Yaskawa INFORM job: R2_W53-A5(180,0)AWOK.JBI

/JOB
//NAME R2_W53-A5(180,0)AWOK
///FOLDERNAME AWOK
//POS
///NPOS 32,32,0,2,0,0
///TOOL 0
///POSTYPE PULSE
///PULSE
C00000=78189,-67986,-96830,-10467,37806,-7797
C00001=92440,-137165,-107216,-20191,-1154,-30432
C00002=105503,-62969,-89657,-20228,86421,-49842
C00003=110518,-93811,-72284,-25294,103379,-67006
C00004=109543,-97011,-70118,-25208,100377,-66720
C00005=109125,-98154,-69170,-25203,99187,-66619
C00006=109125,-97062,-67033,-25140,98501,-66471
C00007=109125,-98154,-69170,-25203,99187,-66619
C00008=109271,-97171,-69065,-25206,99632,-66661
C00009=108845,-100765,-70348,-25219,98541,-66586
C00010=109271,-97171,-69065,-25206,99632,-66661
C00011=102810,-100484,-71733,-21889,96863,-67504
C00012=105287,-101169,-71975,-21344,97318,-66684
C00013=102810,-100484,-71733,-21889,96863,-67504
C00014=103151,-99431,-72768,-21891,98051,-67597
C00015=103951,-96443,-75155,-21958,101060,-67861
C00016=107257,-100648,-73272,-10850,107469,-69930
C00017=107258,-98768,-69563,-10763,106175,-69811
C00018=112732,-102414,-73458,-8827,107350,-67938
C00019=107259,-98817,-69673,-10765,106216,-69815
C00020=107581,-95618,-67198,-10659,106378,-69713
C00021=107132,-98744,-68135,-10755,105306,-69778
C00022=106572,-95477,-62214,-34043,93376,-79177
C00023=105781,-95731,-62292,-31308,97836,-75763
C00024=108056,-94926,-62112,-24163,105722,-68769
C00025=107208,-94572,-61089,-27775,101795,-84365
C00026=107266,-95021,-62493,-27833,102377,-84485
C00027=107266,-96693,-65652,-27971,103342,-84724
C00028=122843,-112109,-94588,-24450,117159,-81729
C00029=129835,-134677,-103725,-23924,94621,-78436
C00030=118025,-147103,-122296,-20754,32567,-81607
C00031=61610,-147103,-122296,-20754,32567,-81607
BC00000=191480,239490,1075165
BC00001=211047,195744,1075167
BC00002=219137,147036,1075169
BC00003=237082,38982,1075175
BC00004=237082,38982,1075175
BC00005=237082,38982,1075175
BC00006=237082,38982,1075175
BC00007=237082,38982,1075175
BC00008=237082,38982,1075175
BC00009=237082,38982,1075175
BC00010=237082,38982,1075175
BC00011=237082,38982,1075175
BC00012=237082,38982,1075175
BC00013=237082,38982,1075175
BC00014=237082,38982,1075175
BC00015=237082,38982,1075175
BC00016=264111,22038,1075175
BC00017=262937,27424,1075175
BC00018=262467,29578,1075175
BC00019=262467,29578,1075175
BC00020=262467,29578,1075175
BC00021=262467,29578,1075175
BC00022=226039,41359,1075175
BC00023=234841,33538,1075175
BC00024=257071,26439,1075171
BC00025=249909,32280,1075175
BC00026=249045,29914,1075175
BC00027=246884,23997,1075175
BC00028=246884,23997,1075175
BC00029=246884,23997,1075175
BC00030=246884,78765,1075175
BC00031=208302,298254,1075175
///POSTYPE BASE
///RECTAN
///RCONF 0,0,0,0,0,0,0,0,0,0,0,0,0,0,0,0,0,0,0,0,0,0,0,0
P00006=0.222,-3.123,-1.508,0.0000,0.0000,0.0000
P00023=0.143,-0.036,0.682,0.0000,0.0000,0.0000
//INST
///DATE 2023/11/16 10:54
///ATTR SC,RW
///GROUP1 RB1,BS1
NOP
'r2_W53-A5(180,0)
'Path S1074
MOVJ C00000 BC00000 VJ=20.00
SFTOF
MOVJ C00001 BC00001 VJ=20.00
MOVJ C00002 BC00002 VJ=20.00
MOVJ C00003 BC00003 VJ=20.00
MOVL C00004 BC00004 V=100.0
MOVL C00005 BC00005 V=60.0
REFP 3 C00006 BC00006
CALL JOB:SEARCH-R1
SET P023 P006
SFTON P023
MOVL C00007 BC00007 V=60.0
MOVL C00008 BC00008 V=60.0
REFP 3 C00009 BC00009
CALL JOB:SEARCH-R1
SET P023 P006
SFTON P023
MOVL C00010 BC00010 V=60.0
MOVL C00011 BC00011 V=60.0
REFP 3 C00012 BC00012
CALL JOB:SEARCH-R1
SET P023 P006
SFTON P023
MOVL C00013 BC00013 V=60.0
MOVL C00014 BC00014 V=100.0
MOVL C00015 BC00015 V=100.0
'Path W1075
SFTOF
MOVJ C00016 BC00016 VJ=20.00
MOVL C00017 BC00017 V=100.0
SFTON P023
MOVL C00018 BC00018 V=100.0 PL=0
REFP 1 C00019 BC00019
REFP 2 C00020 BC00020
MACRO1 MJ#(0) ARGF9
ARCON
MOVL C00021 BC00021 V=10.0
MOVL C00022 BC00022 V=10.0
MOVL C00023 BC00023 V=10.0
MOVL C00024 BC00024 V=10.0
MOVL C00025 BC00025 V=10.0
ARCOF
MOVL C00026 BC00026 V=100.0
MOVL C00027 BC00027 V=100.0
MOVJ C00028 BC00028 VJ=20.00
MOVJ C00029 BC00029 VJ=20.00
MOVJ C00030 BC00030 VJ=20.00
MOVJ C00031 BC00031 VJ=20.00
SFTOF
END
